FUNCTION_BLOCK FB_BatterySupply EXTENDS RACBaseObjects.FB_Machine
VAR_INPUT
	bSafetyBoxPlace_permissive			: BOOL;
	
	bPlace_MaterialRequest				: BOOL;
END_VAR
VAR_OUTPUT
	bSafetyBoxPlace_OutOfZone			: BOOL;
	
	sPieceSN							: STRING;
	sPieceOnGantrySN					: STRING;
	sPieceOnSliderSN					: STRING;
	
	bPlace_Done							: BOOL;
END_VAR
VAR
	fbTrayFeeder						: RACBaseObjects.FB_TrayFeeder;
	fbRobot								: RACBaseObjects.FB_Robot;
	fbScanner							: RACBaseObjects.FB_Scanner;
	
	// Auto procees is scanning
	bScann								: BOOL;
	
	// Auxiliar bool array for reject places inputs
	bAvailableNests						: ARRAY[0..7] OF BOOL;
END_VAR

SUPER^.MachineMain();
//	Tray Feeder instance
	fbTrayFeeder(						sDeviceID:=	'',
										bStopExecution:=bStopExecution,
										bAlarmReset:=bAlarmReset,
										diStationState:=diStationState,
										bInit_StartPermissive:=fbRobot.bInit_Finished,
										bSafetyBoxDeliver_permissive:=fbRobot.bSafetyBoxPick_OutOfZone,
										bChangeTrayRequest:=fbRobot.bPick_AllMaterialPicked);

//	Robot instance
//	fbRobot(							sDeviceID:=	'',
//										bStopExecution:=bStopExecution,
//										bAlarmReset:=bAlarmReset,
//										diStationState:=diStationState,
//										bInit_StartPermissive:=bInit_StartPermissive,
//										bSafetyBoxPick_Permissive:=fbTrayFeeder.bSafetyBoxDeliver_isSafe,
//										bSafetyBoxPlace_Permissive:=bSafetyBoxPlace_permissive,
//										bSafetyBoxReject_Permissive:=FALSE,
//										bOKMaterialReadyToPick:=fbTrayFeeder.bMaterial_ReadyToPick,
//										bNGMaterialReadyToPick:=FALSE,
//										bPiceIsGood:=TRUE,
//										bPiceIsNG:=FALSE,
//										bPlace_MaterialRequest:=bPlace_MaterialRequest,
//										bReject_MaterialRequest:=bAvailableNests,
//										bSafetyBoxPlace_OutOfZone=>bSafetyBoxPlace_OutOfZone,
//										bPlace_Done=>bPlace_Done);

//	Scanner insance
	fbScanner(							sDeviceID:=	'',
										bStopExecution:=bStopExecution,
										bAlarmReset:=bAlarmReset,
										bIn_Trigger:=bScann,
										bDisable:=FALSE,
										iTotalRetries:=2,
										Timeout:=t#1s);

METHOD Alarm
sAlarm:= CONCAT(STR1:=fbTrayFeeder.sAlarm, STR2:=fbRobot.sAlarm);
sAlarm:= CONCAT(STR1:=sAlarm,STR2:=fbScanner.sAlarm);
END_METHOD

METHOD Auto
VAR
END_VAR
//	When slider is not taking piece, reaching delivery position or delivering unit, clear piece on slider code var
	IF (fbTrayFeeder.diActualSeqStep<>1110) AND (fbTrayFeeder.diActualSeqStep<>1120) AND (fbTrayFeeder.diActualSeqStep<>1130) THEN
		sPieceSN:='';
	END_IF

//	When finish reading save the code in a var
	IF fbTrayFeeder.diActualSeqStep=1110 THEN
		bScann:=TRUE;
		IF (fbScanner.bCompleted) AND (sPieceSN<>fbScanner.sCode) THEN
			sPieceSN:=fbScanner.sCode;
		END_IF
	END_IF

//	When gantry takes the battery translate last serial code readed
	IF (fbTrayFeeder.diActualSeqStep=1130) AND (sPieceOnGantrySN=sPieceSN) THEN
		sPieceOnGantrySN:=sPieceSN;
	END_IF

//	When gantry release the battery translate serial code to other var
	IF (fbTrayFeeder.diActualSeqStep=1150) AND (sPieceOnSliderSN<>sPieceOnGantrySN) THEN
		sPieceOnSliderSN:=sPieceOnGantrySN;
	END_IF
END_METHOD

METHOD Init
bInit_Finished:=fbTrayFeeder.bInit_Finished AND fbRobot.bInit_Finished AND fbScanner.bConnected;
END_METHOD

METHOD IO
//	For robot available places inputs
	bAvailableNests[0]					:= FALSE;
	bAvailableNests[1]					:= FALSE;
	bAvailableNests[2]					:= FALSE;
	bAvailableNests[3]					:= FALSE;
	bAvailableNests[4]					:= FALSE;
	bAvailableNests[5]					:= FALSE;
	bAvailableNests[6]					:= FALSE;
	bAvailableNests[7]					:= FALSE;
END_METHOD

{warning 'Add method implementation '}
METHOD Manual
END_METHOD

{warning 'Add method implementation '}
METHOD Pause
END_METHOD

{warning 'Add method implementation '}
METHOD Stop
END_METHOD

END_FUNCTION_BLOCK

(* stored: Version 1.1.0.1, ProductVersion 3.1.4024.12
   POU FB_BatterySupply: Id {174d994e-be67-4f6e-9f61-9168120df54b}, SpecialFunc None
   Method Alarm: Id {92f8f847-4bbb-49b0-90c0-ee4d6ac5ad7f}
   Method Auto: Id {4f5384bf-b44f-4a01-b54d-42ab93e4da30}
   Method Init: Id {475a2b99-ca25-417d-a341-935d7671e03c}
   Method IO: Id {dfc4259a-e026-4b8f-a3b5-16afbaddf784}
   Method Manual: Id {d94dba60-c477-4bbe-804a-c4c2d515ccef}
   Method Pause: Id {3a21d47f-efff-43d9-afa2-98570106cfcd}
   Method Stop: Id {c711b130-f538-4384-b6ab-46945978c516} *)
